PROGRAM Conc
VAR
END_VAR

// NETWORK 1

END_PROGRAM

(* stored: Version 1.1.0.1, ProductVersion 3.1.4024.12
   POU Conc: Id {96ed4091-2a3c-4981-a685-3b97a3982cca}, SpecialFunc None *)
